Staubli VAL3: getNextID.pgx

public program getNextID(num& x_nCamID (dimensions=1), bool& x_bError (dimensions=1))
  local num l_nIndex
  local bool l_bFound
begin
  //-----------------------------------------------------------------------
  //Header begin
  //Description of program
  //  Return an available camera's ID.
  //  By default, maximum  number of camera connected at the same time is 10 (ID 0 to 9)
  //  this can be changed by resizing cCamera array (this array must contain one more element
  //  than the maximum amount of cameras you want to allow).
  //
  //Output parameters
  //  num x_nCamID :
  //    role : camera's ID (only use if no errors returned in x_bError)
  //
  //  bool x_bError :
  //    role : returns true if an error occurred (no more ID available)
  //    and false otherwise, then call get error functions to recuperate
  //    error code / message
  //
  //Examples
  //    call returnID(l_nCamID,l_bError)
  //
  //History
  //  Creation : 15-05-12 - t.caille
  //Header end
  //-----------------------------------------------------------------------

  l_nIndex=0
  l_bFound=false
  //program scan free camera's ID
  do
    if cCamera[l_nIndex].bConnected==false
      x_nCamID=l_nIndex
      l_bFound=true
    endIf
    l_nIndex=l_nIndex+1
  until l_nIndex==size(cCamera)-1 or l_bFound==true
  //No more place for another camera
  if l_nIndex==size(cCamera)-1 and l_bFound==false
    x_bError=true
    x_nCamID=size(cCamera)-1
    nLibErrorCode=201
  endIf
end
